ABB RobotStudio station: test_definition.rsstn

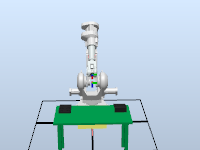
Station IRB2400_MoveJLC_RW6.10.02 (saved by RobotStudio 7.0.8746.631)
Controller 2400-200424, task T_ROB1: task frame (RAPID world) sits at (0, 0, 200) mm in the station
Controller 2400-200424
  mechanical unit ROB_1: IRB2400_16_150__02, 6 joints, base frame (0, 0, 0) mm
Layout (positions relative to the parent item):
  - Stand_H200 [part, from Libraries\RobotBase_H200.rslib]
  - Plate_Flat [part] at (940, -410, 685) mm
  - Plate_Inclined [part] at (935.23, 410, 685) mm
  - Pen_90 [mechanism, from Libraries\Pen_90.rslib] at (700, 0, 1150) mm, rotated rx 0 ry 90 rz 0 deg
  - Table_H685 [part, from Libraries\Table_H685.rslib] at (1100, 0, 0) mm
  - TCP_Teaching_Tool [part, from Libraries\TCP_Teaching_Tool.rslib] at (1100, 0, 685) mm
  - IRB2400_16_150__02 [mechanism, from Robots\IRB2400_16_150_G_02.rslib] at (0, 0, 200) mm; joint values [0, -0.24, 0.6505, 0, -0.6505, 0] (rad or m)
Attachment: Plate_Flat is attached to Table_H685
Attachment: Plate_Inclined is attached to Table_H685
Attachment: Pen_90 is attached to IRB2400_16_150__02 / Link6
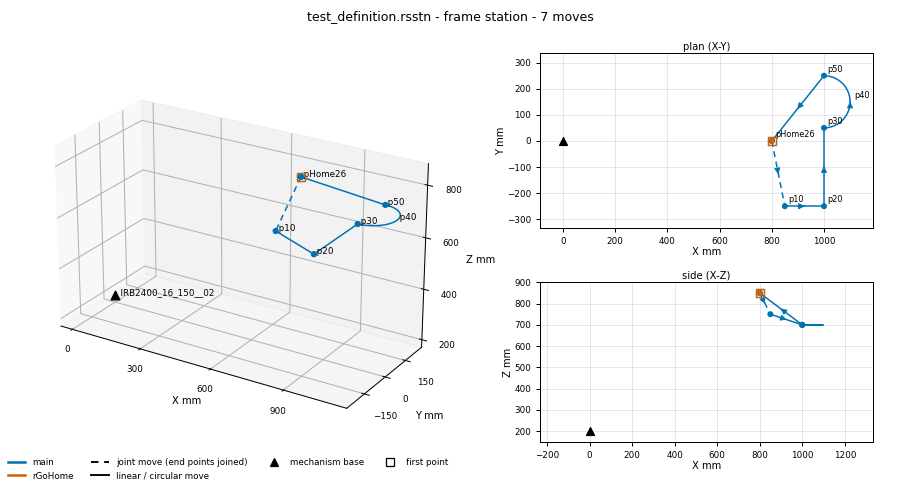
[picture p0: tool path of test_definition.rsstn in frame station, 7 of 9 moves have a stored position in this frame; points joined in program order, loops and branches not executed]
Targets, tools, work objects and paths stored in the station, written as RAPID:
! task T_ROB1
MODULE MainModule
  CONST robtarget p10:=[[850,-250,750],[0.000039112,0.000013788,1,-0.000000552],[-1,-1,0,1],[9E+09,9E+09,9E+09,9E+09,9E+09,9E+09]];
  CONST robtarget p20:=[[1000,-250,700],[0.000039281,0.000013614,1,-0.000000204],[-1,-1,0,1],[9E+09,9E+09,9E+09,9E+09,9E+09,9E+09]];
  CONST robtarget p30:=[[1000,50,700],[0.000040124,0.000014118,1,0.000000242],[0,0,-1,1],[9E+09,9E+09,9E+09,9E+09,9E+09,9E+09]];
  CONST robtarget p40:=[[1100,150,700],[0.000042484,0.000013371,1,0.00000093],[0,0,-1,1],[9E+09,9E+09,9E+09,9E+09,9E+09,9E+09]];
  CONST robtarget p50:=[[1000,250,700],[0.000040967,0.000013858,1,0.000000464],[0,0,-1,1],[9E+09,9E+09,9E+09,9E+09,9E+09,9E+09]];
  PROC main()
    MoveJ pHome26,v300,fine,tPen_90;
    MoveJ p10,v400,fine,tPen_90;
    MoveL p20,v800,fine,tPen_90;
    MoveL p30,v1000,fine,tPen_90;
    MoveC p40,p50,v200,fine,tPen_90;
    MoveL pHome26,v500,fine,tPen_90;
  ENDPROC
ENDMODULE

! task T_ROB1
MODULE COMMON_90R
  TASK PERS wobjdata wobj1:=[FALSE,TRUE,"",[[700,-500,505],[1,0,0,0]],[[0,0,0],[1,0,0,0]]];
  TASK PERS wobjdata wobj2:=[FALSE,TRUE,"",[[694.824,320,504.314],[0.991444758,0,-0.130526981,0]],[[0,0,0],[1,0,0,0]]];
  PERS tooldata tPen_90:=[TRUE,[[100,0,100],[0.707107,0,0.707107,0]],[1,[3.431,0,56.08],[1,0,0,0],0,0,0]];
  CONST robtarget pHome26:=[[800,0,850],[0,0,1,0],[-1,-1,0,1],[9E+09,9E+09,9E+09,9E+09,9E+09,9E+09]];
  CONST jointtarget jpos10:=[[0,0,0,0,0,0],[9E+09,9E+09,9E+09,9E+09,9E+09,9E+09]];
  CONST jointtarget jpos20:=[[0,0,0,0,-1,0],[9E+09,9E+09,9E+09,9E+09,9E+09,9E+09]];
  PROC rCalibPos()
    MoveAbsJ jpos10,v200,fine,tPen_90;
    MoveAbsJ jpos20,v200,fine,tPen_90;
  ENDPROC
  PROC rGoHome()
    MoveJ pHome26,v500,fine,tPen_90;
  ENDPROC
ENDMODULE

! task T_ROB1
MODULE CalibData
  PERS tooldata tPen_90:=[TRUE,[[100,0,100],[0.707106781,0,0.707106781,0]],[1.5,[3.431,0,56.08],[1,0,0,0],0,0,0]];
ENDMODULE

